FUNCTION_BLOCK PiperModule_Test EXTENDS FB_TestSuite
VAR_INPUT
END_VAR
VAR_OUTPUT
END_VAR
VAR
END_VAR

// Copyright (c) 2024 Loupe (https://loupe.team), provided under the MIT License.

END_FUNCTION_BLOCK

(* stored: Version 1.1.0.1
   POU PiperModule_Test: Id {938c15c7-47ae-07e3-18c2-da354fdb321f}, SpecialFunc None *)
